Staubli VAL3: moveGate.pgx

program moveGate()
begin
  movej(gatePosition,flange,mFastMov)
  waitEndMove()
  message="moveGate:done"
  taskCreate "sendStatus",100,sendStatus()
  taskKill("moveGate")
end
